//-----------------------------------------------------------------------------------------------------
//																
//									 	Tkmatik sp. z o.o.
//
//	Name				:		FB_IfmIoLinkRfid
//  Author				:		AM
//	Release Date		:		06.07.2022
//  Current ver			:		v 0.1
// 	Last correction 	:		06.07.2022
// 
//	Description			:						
//	This functional block operate with IFM RFID reader (for example DTI515), connected to PLC via IOLink
//	Allow user to read USER data from RFID tags.
//	1) bReadEnable = true enable asyncronious RFID reading. When DATA is readed FB set bCodeReaded until
//	tag is in reading zone, readed code saved into aReadCode. 
//	bCodeReaded set true if readed code <> last readed code
//	2) For writ USER data to tag: set new code into aWriteCode, than set bWriteEnable = true
//	When system set bWriteDone, code has been writed into tag, bWriteDone resets when bWriteEnable = false
//	4) aIoLinkInputData, bIoLinkTagPresent, nIoLinkErrorValue, bIoLinkCmdEnd, nIoLinkDataCounterIn,
//  bIoLinkCmdStartAck must be connected to IOLink IN; bIoLinkCmdStart, nIoLinkCmmandValue, nIoLinkDataCounter
//	nIoLinkDataCounter must be connecter do IOLink OUT
//
//	Requared hardware	:
//	IFM DTE515 (or other IFM), connected to IOLink
//
//-----------------------------------------------------------------------------------------------------

FUNCTION_BLOCK FB_IfmIoLinkRfid
VAR_INPUT
	//Commands
	bReadEnable						:		BOOL;					//Enable reading USER tag -> aReadCode
	bWriteCmd						:		BOOL;					//Command write aWriteData -> USER tag 
	//Data
	diWriteData						:		DINT;

	//IOLink connection
	aIoLinkInputData  			: 		ARRAY[0..27] OF USINT;
	bIoLinkTagPresent			:		BOOL;
	nIoLinkErrorValue			:		BYTE;
	bIoLinkCmdEnd				:		BOOL;
	nIoLinkDataCounterIn		:		BYTE;
	bIoLinkCmdStartAck			:		BOOL;
	
	
END_VAR

VAR_OUTPUT
	//States and out data
	bCodeReaded						:		BOOL;					//Flag tag on reader 
	bNewCodeReaded					:		BOOL;					//Flag NEW tag on reader
	bWriteCycleEnd					:		BOOL;					//Flag write operation done
	bBysy							:		BOOL;					//Reading or writing operation in process
	diReadedCode					:		DINT;
	bError							:		BOOL;					//RFID sensor error			
	sErrorDescription				:		STRING;					//Error description via Manual
	
	//IOLink connection
	bIoLinkCmdStart				:		BOOL;
	nIoLinkCmmandValue			:		BYTE;
	nIoLinkDataCounterOut		:		BYTE;
	aIoLinkOutputData  			: 		ARRAY[0..27] OF USINT;
END_VAR

VAR
	fbDIntTo4Byte					:		FB_DIntTo4Byte;
	aWriteData						:		ARRAY[0..15] OF BYTE;	//User data for writing	
	nWriteLengthLo					:		BYTE:=4;					//Length ou user data (max = 16)
	
	aReadCode						:		ARRAY [0..15] OF BYTE;	//Readed code value (saved)

	
	i								:		INT;					//FOR iterator
	
	//Read variables
	aReadCodeOld					:		ARRAY [0..15] OF BYTE;	//Readed code value (saved)
	rtReadFlag						:		R_TRIG;					//Tag on sensor trig
	iRead							:		INT;					//Read cycle case
	
	//Write variables
	iWrite							:		INT;					//Write cycle case
	rtWriteCmd						:		R_TRIG;					//New write command
	ftWriteCmd						:		F_TRIG;					//Write command off (for reset DONE signal)
END_VAR

VAR CONSTANT
	//Config
	nRegUserTagAdressHi				:		INT		:= 2;			//See user's manual
	nRegUserTagAdressLo				:		INT		:= 3;		    //See user's manual
	nRegUserTagLengthHi				:		INT		:= 4;			//See user's manual
	nRegUserTagLengthLo				:		INT		:= 5;		    //See user's manual
	nWriteLengthHi					:		BYTE	:= 0;			//We use only first 16 byte of tag

	//Operations
	nNoOperationCommand				:		BYTE	:= 16#04;		//Value of command register NOP
	nWriteUserDataCommand			:		BYTE	:= 16#04;		//Value of command register WR
	nReadUserDataCommand			:		BYTE	:= 16#01;		//Value of command register RD
	nBaseUserTagAdreessHi			:		BYTE	:= 16#00;		//Defaul adress of User data, we use only max first 16 byte;
	nBaseUserTagAdreessLo			:		BYTE	:= 16#00;		//Defaul adress of User data, we use only max first 16 byte;
END_VAR

aErrorHandling();
aMain();

ACTION aErrorHandling:
bError		 							:= nIoLinkErrorValue >0;

CASE nIoLinkErrorValue OF

	16#00	:	sErrorDescription		:= '';
	16#01	:	sErrorDescription		:= 'RFID UNKNOWN COMMAND';
	16#11	:	sErrorDescription		:= 'COMMAND NO RESPONSE';
	16#12	:	sErrorDescription		:= 'COMMAND RX ERROR';
	16#21	:	sErrorDescription		:= 'TAG COMMAND NOT SPECIFIED';
	16#22	:	sErrorDescription		:= 'TAG COMMAND SYNTAX';
	16#23	:	sErrorDescription		:= 'TAG OPTION NOT SUPPORTED';
	16#2F	:	sErrorDescription		:= 'TAG OTHER ERROR';
	16#30	:	sErrorDescription		:= 'TAG BLOCK NOT USABLE';
	16#31	:	sErrorDescription		:= 'TAG BLOCK ALREADY BLOCKED';
	16#32	:	sErrorDescription		:= 'TAG BLOCK NOT UPDATEBLE';
	16#33	:	sErrorDescription		:= 'TAG BLOCK WRITE VERIFY';
	16#34	:	sErrorDescription		:= 'TAG BLOCK LOCK VERIFY';
	ELSE
		sErrorDescription				:= 
			CONCAT(STR1 				:= 'UNKNOWN ERROR CODE = 0x',
				   STR2 				:= BYTE_TO_HEXSTR(in:=nIoLinkErrorValue,iPrecision:=2,bLoCase:=TRUE));
END_CASE
END_ACTION

ACTION aMain:
IF (iRead = 0 AND iWrite = 0) THEN
	bIoLinkCmdStart						:= FALSE;
	nIoLinkCmmandValue					:= nNoOperationCommand;
END_IF

//Read operations
IF (bReadEnable AND iWrite = 0 AND iRead = 0) THEN
	iRead								:= 1;
END_IF

//Write operation
rtWriteCmd(CLK:=bWriteCmd);
ftWriteCmd(CLK:=bWriteCmd);
IF (rtWriteCmd.Q AND iWrite = 0 AND iRead=0) THEN
	iWrite								:= 1;
END_IF
IF ftWriteCmd.Q THEN
	bWriteCycleEnd						:= FALSE;
	iWrite 								:= 0;
END_IF

//Actions calling
aWrite();
aRead();

bBysy									:=	iRead > 0 OR iWrite > 0;
END_ACTION

ACTION aRead:
CASE iRead OF
	0:
		;
	1:
		bIoLinkCmdStart					:= FALSE;
		iRead							:= 2;
	2:
		nIoLinkCmmandValue	 			:= nReadUserDataCommand; // read user data
		bIoLinkCmdStart					:= TRUE;
		iRead							:= 3;
	3:
		rtReadFlag(CLK := (bIoLinkTagPresent AND bIoLinkCmdEnd));
		
		IF (rtReadFlag.Q) THEN
			FOR i:=0 TO 15 DO
		
				IF (aReadCode[i] <> USINT_TO_BYTE( aIoLinkInputData[i])) THEN
					bNewCodeReaded		:= TRUE;
				END_IF
		
				aReadCode[i] 			:= USINT_TO_BYTE( aIoLinkInputData[i]);
		
			END_FOR
			diReadedCode				:=	DWORD_TO_DINT(F_4BYTES_TO_DWORD(BByte0:=aReadCode[3],BByte1:=aReadCode[2],BByte2:=aReadCode[1],BByte3:=aReadCode[0]));
				
			//iReadedCode					:= F_2Bytes_To_Word(byHigh:=aReadCode[4],byLow:=aReadCode[3]); 
		END_IF

		bCodeReaded  							:= bIoLinkTagPresent AND bIoLinkCmdEnd;

		IF (NOT bCodeReaded) THEN
			bNewCodeReaded						:= FALSE;
		END_IF
		
		IF (NOT bReadEnable) THEN
			FOR i:=0 TO 15 DO
				aReadCodeOld[i]					:= 0;
			END_FOR
			bCodeReaded							:= FALSE;
			bNewCodeReaded						:= FALSE;
			iRead								:= 0;
		END_IF
END_CASE
END_ACTION

ACTION aWrite:
CASE iWrite OF
	0:
		;
	1:
		IF (bIoLinkTagPresent) THEN
			iWrite								:= 2;
		END_IF
	2:
		bIoLinkCmdStart							:= FALSE;
		iWrite									:= 3;
	3:
		nIoLinkCmmandValue	 					:= nWriteUserDataCommand;
		
		aIoLinkOutputData[0]					:= 0;
		aIoLinkOutputData[1]					:= 0;
		
		aIoLinkOutputData[nRegUserTagAdressHi]	:= nBaseUserTagAdreessHi;
		aIoLinkOutputData[nRegUserTagAdressLo]	:= nBaseUserTagAdreessLo;
		aIoLinkOutputData[nRegUserTagLengthHi]	:= nWriteLengthHi;
		aIoLinkOutputData[nRegUserTagLengthLo]	:= nWriteLengthLo;
		
		aIoLinkOutputData[6]					:= 0;
		aIoLinkOutputData[7]					:= 0;
		aIoLinkOutputData[8]					:= 0;
		aIoLinkOutputData[9]					:= 0;
		aIoLinkOutputData[10]					:= 0;
		aIoLinkOutputData[11]					:= 0;
		aIoLinkOutputData[12]					:= 0;
		aIoLinkOutputData[13]					:= 0;
		aIoLinkOutputData[14]					:= 0;
		aIoLinkOutputData[15]					:= 0;
		aIoLinkOutputData[16]					:= 0;
		aIoLinkOutputData[17]					:= 0;
		aIoLinkOutputData[18]					:= 0;
		aIoLinkOutputData[19]					:= 0;
		aIoLinkOutputData[20]					:= 0;
		aIoLinkOutputData[21]					:= 0;
		aIoLinkOutputData[22]					:= 0;
		aIoLinkOutputData[23]					:= 0;
		aIoLinkOutputData[24]					:= 0;
		aIoLinkOutputData[25]					:= 0;
		aIoLinkOutputData[26]					:= 0;

		nIoLinkDataCounterOut					:= 0;
		bIoLinkCmdStart							:= TRUE;
		iWrite									:= 4;
	4:
		IF (bIoLinkCmdStartAck) THEN
			iWrite								:= 5;
		END_IF
	5:
		fbDIntTo4Byte(iInput:=diWriteData,by0=>aWriteData[0],by1=>aWriteData[1],by2=>aWriteData[2],by3=>aWriteData[3]);

		FOR i:=0 TO (nWriteLengthLo-1) DO
			aIoLinkOutputData[i]				:= aWriteData[i];
		END_FOR
		FOR i:=nWriteLengthLo TO 26 DO
			aIoLinkOutputData[i]				:= 0;
		END_FOR
		nIoLinkDataCounterOut					:= 1;
		iWrite									:= 6;
	6:
		IF (nIoLinkDataCounterIn = 1) THEN
			iWrite								:= 7;
		END_IF
	7:
		IF (bIoLinkCmdEnd) THEN
			iWrite									:= 0;	
			bWriteCycleEnd							:= TRUE;
		END_IF	
END_CASE
END_ACTION

END_FUNCTION_BLOCK

(* stored: Version 1.1.0.1, ProductVersion 3.1.4026.13, FileIdentifier 0b48d218d20321862a4d017e14f57cd1d2232a92, FileSignature 33fee9548153f79941ba2747c623bd2834359df244e46d2612b28fa8df9504291dc3a417fc1d38a0df8c2cc05a9f04a339c6e63524aa94e46f7a56ea93a97b5e83fda143c172ff206a41a65ff6b6924a14e81ce7dcd19b78e4ad6a1eafb726556608e96ace3b30cab9476e2c784c6720fc3401008cb88806351d67e044f4986bb25da4a8487b527deb2bf42ac8b2f7ff2e900f9b0ee48d1d23fadde7e427ae570e9a9de6e5231b33ee8e82b30cfa7757c7068c67e18846b5a25b3aaf0cb39d3730db6929dfe43846487f1f5f59b9f174dee7058dbec1ed75839d09f9fe9a8357a19ae66b778a4aac809fd5500c7549fd9544b42e8d6b8673d1178d3345c771c3
   POU FB_IfmIoLinkRfid: Id {d0480aea-5672-4141-b189-c2f2f9dc9946}, SpecialFunc None
   Action aErrorHandling: Id {017ac3fd-83b8-4898-a3cf-b04780a7cd65}
   Action aMain: Id {e5d5bf13-439a-447e-947e-c760ed70322c}
   Action aRead: Id {6fe714a6-7e8d-4da6-ad8d-d33691a4253c}
   Action aWrite: Id {8b48c26d-9645-422b-b9d3-96eaaf184840} *)
